PROGRAM MAIN
VAR
	_BOOL_TestSuite : _BOOL_TestSuite;
END_VAR

TcUnit.RUN();

END_PROGRAM

(* stored: Version 1.1.0.1, ProductVersion 3.1.4024.12
   POU MAIN: Id {7bf63626-4b20-4fda-b93b-546e8359a2c5}, SpecialFunc None *)
